(* PLC project CoDeSys External Library Template, WAGO e!COCKPIT e!COCKPIT, author 3S - Smart Software Solutions GmbH *)
(* stored: creationDateTime 2019-10-29T12:37:19.9762755, version 3.5.5.30, modificationDateTime 2019-10-29T12:36:39.3744516, organization 3S - Smart Software Solutions GmbH *)
(* Library project template with all possible element types, docu and a sample project structure *)

FUNCTION fnZapiszKomunikat : BOOL
  VAR_INPUT
    sCalyKomunikat : alSTRINGKomunikat;
    sTypKomunikatu : STRING;
    sMnemonik : STRING;
    sMACAdres : STRING;
    sIdNadawcy : STRING;
    sIdOdbiorcy : STRING;
    sDaneZapasowe : STRING;
    sDane : alSTRINGKomunikat;
    intTablicaKomunikatowRozmiar : INT;
  END_VAR
  VAR_IN_OUT
    intTablicaKomunikatowZnacznikZapisu : INT;
    arTablicaKomunikatow : alARRAYTablicaKomunikatow;
    sWyslanyKomunikat : alSTRINGKomunikat;
  END_VAR
  VAR
    sKomunikat : alSTRINGKomunikat;
    intBlad : INT;
    typKomunikat : typKomunikat;
  END_VAR

            (* blok do zapisu nowego komunikatu w buforze do wysłania*)

IF sCalyKomunikat = '' THEN
	typKomunikat.sZnacznik := 'ˆ';
	typKomunikat.sTypKomunikatu := sTypKomunikatu;
	typKomunikat.sMnemonikWlasciciela := LEFT(sMnemonik , 3);
	typKomunikat.sMnemonikWlascicielaExt := Right(sMnemonik , 1);
	typKomunikat.sMACAdres := sMACAdres;
	typKomunikat.sIDZrodla := sIdNadawcy;
	typKomunikat.sIDPrzeznaczenia := sIdOdbiorcy;
	typKomunikat.sRezerwa := sDaneZapasowe;
	typKomunikat.sDane := sDane;
	fnKomunikatInOut(	xStringNaStrukture := FALSE ,
						xStringUpdateZeStruktury := FALSE ,
						xStrukturyNaString := TRUE ,
						xWyczyscStrukture := FALSE ,
						xAktualizujZnacznikCzasu := TRUE ,
						xAktualizujDlugoscDanych := TRUE ,
						sKomunikat := sKomunikat ,
						typKomunikat := typKomunikat ,
						intBlad := intBlad);
	ELSE
	sKomunikat := sCalyKomunikat;
END_IF
fnTablicaKomunikatowInkrementacja(intWskaznik := intTablicaKomunikatowZnacznikZapisu , intRozmiarTablicy := intTablicaKomunikatowRozmiar);
arTablicaKomunikatow[intTablicaKomunikatowZnacznikZapisu] := sKomunikat;
sWyslanyKomunikat := sKomunikat;

          
END_FUNCTION
